# EPICS substitutions: epics/db/EK1100.substitutions
# No WcState
#file "./db/ecSlave.template"
#{
#  pattern {}
#          {}
#}

file "./db/EK11X0.template"
{
  pattern {}
          {}
}
